TYPE Room_Ctx_Io :
STRUCT
	in		: Heating_Ctx_Io_In;
	out		: Heating_Ctx_Io_Out;
END_STRUCT
END_TYPE

(* stored: Version 1.1.0.1
   DUT Room_Ctx_Io: Id {67371870-bd5d-49c5-aa16-53adf3c88038} *)
